{region '#Template'}
	{attribute 'Version' := '1.0.0.0'}
	{attribute 'Tags' := '"LCID": "1031", "Text": "Universal, Sensor, AI"'}
	{attribute 'Tags' := '"LCID": "1033", "Text": "Universal, Sensor, AI"'}
	{attribute 'Description' := '"LCID": "1031", "Text": "AI mit IO"'}
	{attribute 'Description' := '"LCID": "1033", "Text": "AI with IO"'}
{endregion}	 
FUNCTION_BLOCK FB_BA_SensorAnalog_IO EXTENDS FB_BA_View
VAR_INPUT
END_VAR
VAR_INPUT CONSTANT
	MV					: FB_BA_AI_IO;		
END_VAR
VAR_OUTPUT
	fPresentValue		: REAL;
	bEvent				: BOOL;
	eEventState			: E_BA_EventState;	
END_VAR
VAR
END_VAR

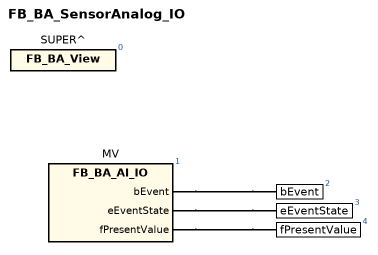
SUPER^(); // FB_BA_View
MV(); // FB_BA_AI_IO
bEvent := MV.bEvent;
eEventState := MV.eEventState;
fPresentValue := MV.fPresentValue;

METHOD FB_init : BOOL
VAR_INPUT
	bInitRetains : BOOL; // if TRUE, the retain variables are initialized (warm start / cold start)
	bInCopyCode : BOOL;  // if TRUE, the instance afterwards gets moved into the copy code (online change)
END_VAR
MV.iParent						:= THIS^;		
MV.iLabel 						:= LblUniFieldDevice.SensorAnalog_MV;
MV.sObjectName					:= '{Idx=01}';
MV.sDeviceType					:= '';
MV.bEnOutOfService				:= FALSE;
MV.eUnit						:= E_BA_Unit.eTemperature_DegreesCelsius;
MV.fResolution 					:= 0.01;
MV.fScaleOffset 				:= 0; 	
MV.fCOVIncrement				:= BA2_Param.fDefCOVIncrement;
MV.nEventClassID				:= EventClasses.AlarmTechnicalExtended;
MV.stTimeDelay.nToNormal		:= BA2_Param.nDefTimeDelay_ToNormal;
MV.stTimeDelay.nToAbnormal		:= BA2_Param.nDefTimeDelay_ToAbnormal;
MV.stHighLimit.bEnable			:= FALSE;
MV.stHighLimit.fValue			:= 0.0;		
MV.stLowLimit.bEnable			:= FALSE;
MV.stLowLimit.fValue			:= 0.0;
MV.fLimitDeadband 				:= BA2_Param.fDefLimitDeadband;
MV.bAcknowledgeRm				:= FALSE;	
MV.aEventTransitionText[1]		:= txtEvent_Exceeded;
MV.aEventTransitionText[2]		:= txtEvent_Disturb;
MV.aEventTransitionText[3]		:= txtEvent_Normal;
MV.bEventDetectionEnable		:= TRUE;
MV.eEnPlantLock					:= E_BA_LockPriority.eNoLock;
END_METHOD

END_FUNCTION_BLOCK

(* stored: Version 1.1.0.1, ProductVersion 3.1.4024.9
   POU FB_BA_SensorAnalog_IO: Id {2b8cd12e-a1b5-4f20-ba20-fd72580da6ca}, SpecialFunc None
   Method FB_init: Id {fd02f8b1-ae19-409a-90ef-b7540c363ac2} *)
